# EPICS substitutions: iocs/MC05/db/SAI_IOCsystem.substitutions
# DEVICE: device name
# CARD:
# CS_VERSION_VAL

file /opt/epics/modules/uIOCSystem/db/uIOCsystem.template {
pattern { DEVICE, CARD, CS_VERSION_VAL}
	{ "XF:06BM-OP{MC:05}", "0", "v0.01" }
}

#EOF
